FUNCTION_BLOCK FuseChannelBasic IMPLEMENTS IFuseChannelBasic
VAR_INPUT
END_VAR
VAR_OUTPUT
END_VAR
VAR
	_Chn : EL922x_ChannelBasic;
END_VAR


PROPERTY CoolDownLock : BOOL
GET
CoolDownLock := _Chn.Status.CoolDownLock;
END_GET
END_PROPERTY


PROPERTY CurrentLevelWarning : BOOL
GET
CurrentLevelWarning := _Chn.Status.CurrentLevelWarning;
END_GET
END_PROPERTY


PROPERTY Diag : BOOL
GET
Diag := _Chn.Status.Diag;
END_GET
END_PROPERTY


PROPERTY Enabled : BOOL
GET
Enabled := _Chn.Status.Enabled;
END_GET
END_PROPERTY


PROPERTY Error : BOOL
GET
Error := _Chn.Status.Error;
END_GET
END_PROPERTY


PROPERTY HardwareProtection : BOOL
GET
HardwareProtection := _Chn.Status.HWProtection;
END_GET
END_PROPERTY


METHOD ResetFuse : BOOL
_Chn.Control.Reset := NOT _Chn.Control.Reset;
END_METHOD


PROPERTY StateReset : BOOL
GET
StateReset := _Chn.Status.StateReset;
END_GET
END_PROPERTY


PROPERTY StateSwitch : BOOL
GET
StateSwitch := _Chn.Status.StateSwitch;
END_GET
END_PROPERTY

METHOD SwitchFuse : BOOL
_Chn.Control.Switch := NOT _Chn.Control.Switch;
END_METHOD


PROPERTY Tripped : BOOL
GET
Tripped := _Chn.Status.Tripped;
END_GET
END_PROPERTY


PROPERTY TxPDOState : BOOL
GET
TxPDOState := _Chn.Status.TxPDOState;
END_GET
END_PROPERTY

END_FUNCTION_BLOCK

(* stored: Version 1.1.0.1, ProductVersion 3.1.4024.5
   POU FuseChannelBasic: Id {4ed96906-348d-4332-82b9-9ff251aa9215}, SpecialFunc None
   Property CoolDownLock: Id {e07ba71c-64f0-4e04-b6fd-21df6f2e6640}
   Get Get: Id {fcd1bfbf-f199-46c4-94f7-ada93c449d97}
   Property CurrentLevelWarning: Id {6b5391bf-b097-4229-a006-46d47d6dcc33}
   Get Get: Id {e6fbf675-527c-4bc8-a456-a59280cac53a}
   Property Diag: Id {c19887ed-8941-48ed-a340-c98b9230f87a}
   Get Get: Id {03e95921-a469-49bf-bcc6-3e9f19c43db9}
   Property Enabled: Id {2a46a555-1d99-4c01-ad93-ccc8110336dc}
   Get Get: Id {664d46c7-1dd4-45a1-b349-c5c86c45280e}
   Property Error: Id {b69c5ab8-7941-4552-b193-0be2678d7097}
   Get Get: Id {d1eb32f1-4e46-4491-bd50-cbea8d57b189}
   Property HardwareProtection: Id {b218c2aa-6263-4c61-bd8b-a29143ea2418}
   Get Get: Id {4e4f691c-016e-4a8f-93b7-5e48b1b46d98}
   Method ResetFuse: Id {4099a5a6-cd71-46e5-b9da-e923d8398584}
   Property StateReset: Id {52ce117b-a1fb-4c98-a4a1-0594891cbbb8}
   Get Get: Id {7eb24e15-9220-4e82-82c9-865cbdaaef8b}
   Property StateSwitch: Id {35580279-0886-4256-8167-2e5eed97eb2a}
   Get Get: Id {3162808d-8e41-4291-8829-ece59958aac1}
   Method SwitchFuse: Id {95478f6a-fe56-4906-bd9f-48f1a4d03935}
   Property Tripped: Id {7df8a10e-0996-41a2-b79a-8263c6bc7ceb}
   Get Get: Id {9175f461-459a-4541-84fd-e9aea67edcaa}
   Property TxPDOState: Id {17eb5a53-337b-4b81-a4ea-35d68feba354}
   Get Get: Id {d05317f6-bf25-4646-8393-5b8d9276977a} *)
